INTERFACE I_SubModuleCollection

PROPERTY Count : UDINT
GET
END_GET
END_PROPERTY

METHOD TryGetModule: BOOL
VAR_INPUT
	index : UDINT;
END_VAR
VAR_OUTPUT
	Module : I_PackML_BaseModule;
END_VAR
END_METHOD

END_INTERFACE

(* stored: Version 1.1.0.1, ProductVersion 3.1.4024.12
   Itf I_SubModuleCollection: Id {c41f1912-1b18-4af4-95b4-789074d6dc64}
   Property Count: Id {c47a0ebb-dc0b-401b-814c-fac1521c9cfa}
   Get Get: Id {888b243f-5b25-4a32-8495-1a7b00c78961}
   Method TryGetModule: Id {eb76e488-d8e5-4188-bb45-b6ca6b63f5fb} *)
